# EPICS substitutions: iocBoot/ioc34idc/substitutions/canberra_13.substitutions
file "$(MCA)/mcaApp/Db/simple_mca.db"
{
pattern
{P           M       DTYP           INP         PREC  CHANS}
{34idc:med:   mca1  "asynMCA"   "@asyn(AIM2/1 0)"    3  2048}
{34idc:med:   mca2  "asynMCA"   "@asyn(AIM2/1 1)"    3  2048}
{34idc:med:   mca3  "asynMCA"   "@asyn(AIM2/1 2)"    3  2048}
{34idc:med:   mca4  "asynMCA"   "@asyn(AIM2/2 0)"    3  2048}
{34idc:med:   mca5  "asynMCA"   "@asyn(AIM2/2 1)"    3  2048}
{34idc:med:   mca6  "asynMCA"   "@asyn(AIM2/2 2)"    3  2048}
{34idc:med:   mca7  "asynMCA"   "@asyn(AIM3/1 0)"    3  2048}
{34idc:med:   mca8  "asynMCA"   "@asyn(AIM3/1 1)"    3  2048}
{34idc:med:   mca9  "asynMCA"   "@asyn(AIM3/1 2)"    3  2048}
{34idc:med:   mca10 "asynMCA"   "@asyn(AIM3/2 0)"    3  2048}
{34idc:med:   mca11 "asynMCA"   "@asyn(AIM3/3 1)"    3  2048}
{34idc:med:   mca12 "asynMCA"   "@asyn(AIM3/4 2)"    3  2048}
{34idc:med:   mca13 "asynMCA"   "@asyn(AIM3/2 3)"    3  2048}
{34idc:med:   mca0  "Soft Channel"   ""     3  2048}
}

file "$(MCA)/mcaApp/Db/icb_amp.db"
{
pattern
{P			AMP		PORT}
{34idc:med:	amp1	"icbAmp1"}
{34idc:med:	amp2	"icbAmp2"}
{34idc:med:	amp3	"icbAmp3"}
{34idc:med:	amp4	"icbAmp4"}
{34idc:med:	amp5	"icbAmp5"}
{34idc:med:	amp6	"icbAmp6"}
{34idc:med:	amp7	"icbAmp7"}
{34idc:med:	amp8	"icbAmp8"}
{34idc:med:	amp9	"icbAmp9"}
{34idc:med:	amp10	"icbAmp10"}
{34idc:med:	amp11	"icbAmp11"}
{34idc:med:	amp12	"icbAmp12"}
{34idc:med:	amp13	"icbAmp13"}
}

file "$(MCA)/mcaApp/Db/icb_adc.db"
{
pattern
{P			ADC		PORT}
{34idc:med:	adc1	"icbAdc1"}
{34idc:med:	adc2	"icbAdc2"}
{34idc:med:	adc3	"icbAdc3"}
{34idc:med:	adc4	"icbAdc4"}
}

file "$(MCA)/mcaApp/Db/icb_hvps.db"
{
pattern
{P			HVPS	LIMIT	PORT}
{34idc:med:	hvps1	1000	"icbHvps1"}
}
